# B&R Automation Studio project SuperTrak_Distribution (part 2)

#### HmiWriteParID.st - HmiWriteParID function block
```iecst
(******************************************************************************************
 * Copyright: Bernecker + Rainer
 * Author:  B+R
 * Created:  July 2, 2018/1:30 PM
 ******************************************************************************************
 ******************************************************************************************
 * Version History:
 * ----------------------------------------------------------------------------------------
 * V 1.00.0   July 2, 2018/1:30 PM  First Version
 ******************************************************************************************
 * Description:
 * ----------------------------------------------------------------------------------------
 * July 2, 2018/1:30 PM V1.00.0:
 * This FUNCTION block writes ParIDs TO the SuperTrak.
 * Additionally a parameter save can be executed.
 * The FUB can be connected directly TO a HMI application.
 * The parameter structure AND I/Os can be used inside the visu without extra implementation.
 ******************************************************************************************)

FUNCTION_BLOCK HMIWriteParID

	// Check if function block is enabled
	IF Enable THEN
		//####################################################################################//
		// FUNCTION BLOCK IS ENABLED
		//####################################################################################//

		// Check if error occured to change state
		IF Error THEN
			// Go to state error, to wait for acknowledge
			Internal.Step																	:= HMI_WPAR_STATE_ERROR;
		END_IF;

		//************************************************************************************//
		// Operation
		//************************************************************************************//
		CASE Internal.Step OF
			//--------------------------------------------------------------------------------//
			// Initialize internal parameters
			//--------------------------------------------------------------------------------//
			HMI_WPAR_STATE_INIT:

				// Initialize function block to create a logbook entry
				Internal.ArEventLogWrite.AddData											:= ADR(Internal.AddErrorInfo);
				Internal.ArEventLogWrite.AddDataFormat										:= 1;	// zero-terminated string
				Internal.ArEventLogWrite.AddDataSize										:= SIZEOF(Internal.AddErrorInfo);
				Internal.ArEventLogWrite.ObjectID											:= 'HMIWriteParID';
				Internal.AddErrorInfo														:= '';
				Internal.ArEventLogWrite.OriginRecordID										:= 0;	// don't use origin record
				Internal.ArEventLogWrite.TimeStamp											:= 0;	// use internal time stamp

				Internal.Step																:= HMI_WPAR_STATE_INIT_CHECK_CONFIG;

				//--------------------------------------------------------------------------------//
				// Register function block
				//--------------------------------------------------------------------------------//
			HMI_WPAR_STATE_INIT_CHECK_CONFIG:

				// Check configuration inputs if valid
				IF (ADR(Parameters) > 0) AND
					(ADR(HMILink) > 0) THEN
					// Config OK
					Internal.Status.InitConfigCheckDone										:= TRUE;
					Internal.Step															:= HMI_WPAR_STATE_INIT_REG_FB;
				ELSE
					Internal.Status.InitConfigCheckDone										:= FALSE;
					// Set error
					StatusID																:= HMI_ERR_WRONG_CONFIG;
					Error																	:= TRUE;
				END_IF;

				//--------------------------------------------------------------------------------//
				// Register function block
				//--------------------------------------------------------------------------------//
			HMI_WPAR_STATE_INIT_REG_FB:

				// Check if function block is not registered yet
				IF NOT Internal.Status.FuncitonBlockRegistered THEN
					// Check if StControl instance is present and valid
					IF (HMILink.LibraryStatus.FbID[0] <> 0) AND (HMILink.LibraryStatus.LogBookIdent <> 0) THEN
						// Save logbook ident
						Internal.ArEventLogWrite.Ident										:= HMILink.LibraryStatus.LogBookIdent;
						// Create function block ID
						Internal.Status.FuncitonBlockID										:= HMI_CONFIG_FB_ID_HMIWRITE;
						Internal.Status.FunctionBlockIDIndex								:= 0;
						Internal.Status.FuncitonBlockRegistered								:= TRUE;
						// Create logbook entry
						Internal.AddErrorInfo												:= 'Function block registration successfull';
						Internal.ArEventLogWrite.EventID									:= HMI_SUCC_FB_REGISTRATION;
						// Write logbook entry
						WriteLogbookEntry;
					ELSIF (HMILink.LibraryStatus.LogBookIdent <> 0) THEN
						Internal.AddErrorInfo												:= 'No enabled instance of HMIControl could be found';
						Internal.ArEventLogWrite.EventID									:= HMI_ERR_NO_HMICONTROL_REG;
						// Write logbook entry
						WriteLogbookEntry;
						// Set error
						StatusID															:= HMI_ERR_NO_HMICONTROL_REG;
						Error																:= TRUE;
					ELSE
						// Set error
						StatusID															:= HMI_ERR_NO_HMICONTROL_REG;
						Error																:= TRUE;
					END_IF;
				ELSE
					// Continue
					Internal.Step															:= HMI_WPAR_STATE_INIT_CHECK_PAR;
				END_IF;

				//--------------------------------------------------------------------------------//
				// Check parameters
				//--------------------------------------------------------------------------------//
			HMI_WPAR_STATE_INIT_CHECK_PAR:

				// Save parameters
				Internal.ParametersUsed														:= Parameters;
				Internal.Status.InitParCheckDone											:= TRUE;
				Internal.Step																:= HMI_WPAR_STATE_OPERATION;

				//--------------------------------------------------------------------------------//
				// Operation
				//--------------------------------------------------------------------------------//
			HMI_WPAR_STATE_OPERATION:

				// Set active output
				Active																		:= TRUE;

				// Check configuration inputs if valid
				IF (ADR(Parameters) > 0) AND
					(ADR(HMILink) > 0) THEN
					//:::::::::::::::::::::::::::::::::::::::::::::::::::::::::::::::::::::::::::://
					// Parameter update handling
					// Check if parameters should be updated
					IF Update AND NOT Internal.UpdateOld AND NOT UpdateDone THEN

						// Check if parameters are valid
						IF (Parameters.ParameterNumber <> 0) AND
							(Parameters.SectionID <= HMI_CONFIG_NR_OF_SECTIONS) THEN
							// PARAMTERS ARE VALID
							// copy paramters to internal stucture
							Internal.ParametersUsed												:= Parameters;
							// Set status output that update is done
							UpdateDone															:= TRUE;
						ELSE
							// PARAMTERS ARE INVALID
							IF (Parameters.ParameterNumber = 0) THEN
								Internal.AddErrorInfo											:= 'Parameter ID is invalid';
							ELSIF (Parameters.SectionID > HMI_CONFIG_NR_OF_SECTIONS) THEN
								Internal.AddErrorInfo											:= 'Number of section is invalid';
							END_IF;
							Internal.ArEventLogWrite.EventID									:= HMI_ERR_WRONG_PARAMETER;
							// Write logbook entry
							WriteLogbookEntry;
							// Set error
							StatusID															:= HMI_ERR_WRONG_PARAMETER;
							Error																:= TRUE;
						END_IF;
					ELSIF NOT Update THEN
						UpdateDone																:= FALSE;
					END_IF;

					//:::::::::::::::::::::::::::::::::::::::::::::::::::::::::::::::::::::::::::://
					// Service Channel implementation
					// Check if paramter should be written
					IF WriteUDINT AND NOT(CommandDone) THEN
						// Check if parameters are valid
						IF (Parameters.ParameterNumber <> 0) AND
							(Parameters.SectionID <= HMI_CONFIG_NR_OF_SECTIONS) THEN
							// PARAMTERS ARE VALID
							// copy paramters to internal stucture
							Internal.ParametersUsed												:= Parameters;
							Internal.Status.WriteStatus := SuperTrakServChanWrite(Parameters.SectionID,Parameters.ParameterNumber,Parameters.StartParameterIndex,Parameters.ParameterValueCount,ADR(Parameters.UDINTvalue),SIZEOF(Parameters.UDINTvalue));
							IF Internal.Status.WriteStatus <> 0 THEN
								Internal.AddErrorInfo											:= 'Command was not executed successfully: ';
								Info.ErrorCode													:= Internal.Status.WriteStatus;
								GetErrorCode;
								Internal.ArEventLogWrite.EventID								:= HMI_ERR_CMD_NOT_EXECUTED;
								// Write logbook entry
								WriteLogbookEntry;
								// Set error
								StatusID														:= HMI_ERR_CMD_NOT_EXECUTED;
								Error															:= TRUE;
							ELSE
								CommandDone														:= TRUE;
							END_IF;
						ELSE
							// PARAMTERS ARE INVALID
							IF (Parameters.ParameterNumber = 0) THEN
								Internal.AddErrorInfo											:= 'Parameter ID is invalid';
							ELSIF (Parameters.SectionID > HMI_CONFIG_NR_OF_SECTIONS) THEN
								Internal.AddErrorInfo											:= 'Number of section is invalid';
							END_IF;
							Internal.ArEventLogWrite.EventID									:= HMI_ERR_WRONG_PARAMETER;
							// Write logbook entry
							WriteLogbookEntry;
							// Set error
							StatusID															:= HMI_ERR_WRONG_PARAMETER;
							Error																:= TRUE;
						END_IF;

					ELSIF WriteUINT AND NOT(CommandDone) THEN
							// Check if parameters are valid
							IF (Parameters.ParameterNumber <> 0) AND
								(Parameters.SectionID <= HMI_CONFIG_NR_OF_SECTIONS) THEN
								// PARAMTERS ARE VALID
								// copy paramters to internal stucture
								Internal.ParametersUsed												:= Parameters;
								Internal.Status.WriteStatus := SuperTrakServChanWrite(Parameters.SectionID,Parameters.ParameterNumber,Parameters.StartParameterIndex,Parameters.ParameterValueCount,ADR(Parameters.UINTvalue),SIZEOF(Parameters.UINTvalue));
								IF Internal.Status.WriteStatus <> 0 THEN
									Internal.AddErrorInfo											:= 'Command was not executed successfully: ';
									Info.ErrorCode													:= Internal.Status.WriteStatus;
									GetErrorCode;
									Internal.ArEventLogWrite.EventID								:= HMI_ERR_CMD_NOT_EXECUTED;
									// Write logbook entry
									WriteLogbookEntry;
									// Set error
									StatusID														:= HMI_ERR_CMD_NOT_EXECUTED;
									Error															:= TRUE;
								ELSE
									CommandDone														:= TRUE;
								END_IF;
							ELSE
								// PARAMTERS ARE INVALID
								IF (Parameters.ParameterNumber = 0) THEN
									Internal.AddErrorInfo											:= 'Parameter ID is invalid';
								ELSIF (Parameters.SectionID > HMI_CONFIG_NR_OF_SECTIONS) THEN
									Internal.AddErrorInfo											:= 'Number of section is invalid';
								END_IF;
								Internal.ArEventLogWrite.EventID									:= HMI_ERR_WRONG_PARAMETER;
								// Write logbook entry
								WriteLogbookEntry;
								// Set error
								StatusID															:= HMI_ERR_WRONG_PARAMETER;
								Error																:= TRUE;
							END_IF;

					ELSIF WriteUSINT AND NOT(CommandDone) THEN
						// Check if parameters are valid
						IF (Parameters.ParameterNumber <> 0) AND
							(Parameters.SectionID <= HMI_CONFIG_NR_OF_SECTIONS) THEN
							// PARAMTERS ARE VALID
							// copy paramters to internal stucture
							Internal.ParametersUsed												:= Parameters;
							Internal.Status.WriteStatus := SuperTrakServChanWrite(Parameters.SectionID,Parameters.ParameterNumber,Parameters.StartParameterIndex,Parameters.ParameterValueCount,ADR(Parameters.USINTvalue),SIZEOF(Parameters.USINTvalue));
							IF Internal.Status.WriteStatus <> 0 THEN
								Internal.AddErrorInfo											:= 'Command was not executed successfully: ';
								Info.ErrorCode													:= Internal.Status.WriteStatus;
								GetErrorCode;
								Internal.ArEventLogWrite.EventID								:= HMI_ERR_CMD_NOT_EXECUTED;
								// Write logbook entry
								WriteLogbookEntry;
								// Set error
								StatusID														:= HMI_ERR_CMD_NOT_EXECUTED;
								Error															:= TRUE;
							ELSE
								CommandDone														:= TRUE;
							END_IF;
						ELSE
							// PARAMTERS ARE INVALID
							IF (Parameters.ParameterNumber = 0) THEN
								Internal.AddErrorInfo											:= 'Parameter ID is invalid';
							ELSIF (Parameters.SectionID > HMI_CONFIG_NR_OF_SECTIONS) THEN
								Internal.AddErrorInfo											:= 'Number of section is invalid';
							END_IF;
							Internal.ArEventLogWrite.EventID									:= HMI_ERR_WRONG_PARAMETER;
							// Write logbook entry
							WriteLogbookEntry;
							// Set error
							StatusID															:= HMI_ERR_WRONG_PARAMETER;
							Error																:= TRUE;
						END_IF;

					ELSIF WriteDINT AND NOT(CommandDone) THEN
						// Check if parameters are valid
						IF (Parameters.ParameterNumber <> 0) AND
							(Parameters.SectionID <= HMI_CONFIG_NR_OF_SECTIONS) THEN
							// PARAMTERS ARE VALID
							// copy paramters to internal stucture
							Internal.ParametersUsed												:= Parameters;
							Internal.Status.WriteStatus := SuperTrakServChanWrite(Parameters.SectionID,Parameters.ParameterNumber,Parameters.StartParameterIndex,Parameters.ParameterValueCount,ADR(Parameters.DINTvalue),SIZEOF(Parameters.DINTvalue));
							IF Internal.Status.WriteStatus <> 0 THEN
								Internal.AddErrorInfo											:= 'Command was not executed successfully: ';
								Info.ErrorCode													:= Internal.Status.WriteStatus;
								GetErrorCode;
								Internal.ArEventLogWrite.EventID								:= HMI_ERR_CMD_NOT_EXECUTED;
								// Write logbook entry
								WriteLogbookEntry;
								// Set error
								StatusID														:= HMI_ERR_CMD_NOT_EXECUTED;
								Error															:= TRUE;
							ELSE
								CommandDone														:= TRUE;
							END_IF;
						ELSE
							// PARAMTERS ARE INVALID
							IF (Parameters.ParameterNumber = 0) THEN
								Internal.AddErrorInfo											:= 'Parameter ID is invalid';
							ELSIF (Parameters.SectionID > HMI_CONFIG_NR_OF_SECTIONS) THEN
								Internal.AddErrorInfo											:= 'Number of section is invalid';
							END_IF;
							Internal.ArEventLogWrite.EventID									:= HMI_ERR_WRONG_PARAMETER;
							// Write logbook entry
							WriteLogbookEntry;
							// Set error
							StatusID															:= HMI_ERR_WRONG_PARAMETER;
							Error																:= TRUE;
						END_IF;

					ELSIF WriteINT AND NOT(CommandDone) THEN
						// Check if parameters are valid
						IF (Parameters.ParameterNumber <> 0) AND
							(Parameters.SectionID <= HMI_CONFIG_NR_OF_SECTIONS) THEN
							// PARAMTERS ARE VALID
							// copy paramters to internal stucture
							Internal.ParametersUsed												:= Parameters;
							Internal.Status.WriteStatus := SuperTrakServChanWrite(Parameters.SectionID,Parameters.ParameterNumber,Parameters.StartParameterIndex,Parameters.ParameterValueCount,ADR(Parameters.INTvalue),SIZEOF(Parameters.INTvalue));
							IF Internal.Status.WriteStatus <> 0 THEN
								Internal.AddErrorInfo											:= 'Command was not executed successfully: ';
								Info.ErrorCode													:= Internal.Status.WriteStatus;
								GetErrorCode;
								Internal.ArEventLogWrite.EventID								:= HMI_ERR_CMD_NOT_EXECUTED;
								// Write logbook entry
								WriteLogbookEntry;
								// Set error
								StatusID														:= HMI_ERR_CMD_NOT_EXECUTED;
								Error															:= TRUE;
							ELSE
								CommandDone														:= TRUE;
							END_IF;
						ELSE
							// PARAMTERS ARE INVALID
							IF (Parameters.ParameterNumber = 0) THEN
								Internal.AddErrorInfo											:= 'Parameter ID is invalid';
							ELSIF (Parameters.SectionID > HMI_CONFIG_NR_OF_SECTIONS) THEN
								Internal.AddErrorInfo											:= 'Number of section is invalid';
							END_IF;
							Internal.ArEventLogWrite.EventID									:= HMI_ERR_WRONG_PARAMETER;
							// Write logbook entry
							WriteLogbookEntry;
							// Set error
							StatusID															:= HMI_ERR_WRONG_PARAMETER;
							Error																:= TRUE;
						END_IF;

					ELSIF WriteSINT AND NOT(CommandDone) THEN
						// Check if parameters are valid
						IF (Parameters.ParameterNumber <> 0) AND
							(Parameters.SectionID <= HMI_CONFIG_NR_OF_SECTIONS) THEN
							// PARAMTERS ARE VALID
							// copy paramters to internal stucture
							Internal.ParametersUsed												:= Parameters;
							Internal.Status.WriteStatus := SuperTrakServChanWrite(Parameters.SectionID,Parameters.ParameterNumber,Parameters.StartParameterIndex,Parameters.ParameterValueCount,ADR(Parameters.SINTvalue),SIZEOF(Parameters.SINTvalue));
							IF Internal.Status.WriteStatus <> 0 THEN
								Internal.AddErrorInfo											:= 'Command was not executed successfully: ';
								Info.ErrorCode													:= Internal.Status.WriteStatus;
								GetErrorCode;
								Internal.ArEventLogWrite.EventID								:= HMI_ERR_CMD_NOT_EXECUTED;
								// Write logbook entry
								WriteLogbookEntry;
								// Set error
								StatusID														:= HMI_ERR_CMD_NOT_EXECUTED;
								Error															:= TRUE;
							ELSE
								CommandDone														:= TRUE;
							END_IF;
						ELSE
							// PARAMTERS ARE INVALID
							IF (Parameters.ParameterNumber = 0) THEN
								Internal.AddErrorInfo											:= 'Parameter ID is invalid';
							ELSIF (Parameters.SectionID > HMI_CONFIG_NR_OF_SECTIONS) THEN
								Internal.AddErrorInfo											:= 'Number of section is invalid';
							END_IF;
							Internal.ArEventLogWrite.EventID									:= HMI_ERR_WRONG_PARAMETER;
							// Write logbook entry
							WriteLogbookEntry;
							// Set error
							StatusID															:= HMI_ERR_WRONG_PARAMETER;
							Error																:= TRUE;
						END_IF;

					ELSIF WriteREAL AND NOT(CommandDone) THEN
						// Check if parameters are valid
						IF (Parameters.ParameterNumber <> 0) AND
							(Parameters.SectionID <= HMI_CONFIG_NR_OF_SECTIONS) THEN
							// PARAMTERS ARE VALID
							// copy paramters to internal stucture
							Internal.ParametersUsed												:= Parameters;
							Internal.Status.WriteStatus := SuperTrakServChanWrite(Parameters.SectionID,Parameters.ParameterNumber,Parameters.StartParameterIndex,Parameters.ParameterValueCount,ADR(Parameters.REALvalue),SIZEOF(Parameters.REALvalue));
							IF Internal.Status.WriteStatus <> 0 THEN
								Internal.AddErrorInfo											:= 'Command was not executed successfully: ';
								Info.ErrorCode													:= Internal.Status.WriteStatus;
								GetErrorCode;
								Internal.ArEventLogWrite.EventID								:= HMI_ERR_CMD_NOT_EXECUTED;
								// Write logbook entry
								WriteLogbookEntry;
								// Set error
								StatusID														:= HMI_ERR_CMD_NOT_EXECUTED;
								Error															:= TRUE;
							ELSE
								CommandDone														:= TRUE;
							END_IF;
						ELSE
							// PARAMTERS ARE INVALID
							IF (Parameters.ParameterNumber = 0) THEN
								Internal.AddErrorInfo											:= 'Parameter ID is invalid';
							ELSIF (Parameters.SectionID > HMI_CONFIG_NR_OF_SECTIONS) THEN
								Internal.AddErrorInfo											:= 'Number of section is invalid';
							END_IF;
							Internal.ArEventLogWrite.EventID									:= HMI_ERR_WRONG_PARAMETER;
							// Write logbook entry
							WriteLogbookEntry;
							// Set error
							StatusID															:= HMI_ERR_WRONG_PARAMETER;
							Error																:= TRUE;
						END_IF;

					ELSIF WriteSTRING AND NOT(CommandDone) THEN
						// Check if parameters are valid
						IF (Parameters.ParameterNumber <> 0) AND
							(Parameters.SectionID <= HMI_CONFIG_NR_OF_SECTIONS) AND
							(Parameters.STRINGsize > 0) THEN
							// PARAMTERS ARE VALID
							// copy paramters to internal stucture
							Internal.ParametersUsed												:= Parameters;
							Internal.Status.WriteStatus := SuperTrakServChanWrite(Parameters.SectionID,Parameters.ParameterNumber,Parameters.StartParameterIndex,Parameters.STRINGsize,ADR(Parameters.STRINGvalue),Parameters.STRINGsize);
							IF Internal.Status.WriteStatus <> 0 THEN
								Internal.AddErrorInfo											:= 'Command was not executed successfully: ';
								Info.ErrorCode													:= Internal.Status.WriteStatus;
								GetErrorCode;
								Internal.ArEventLogWrite.EventID								:= HMI_ERR_CMD_NOT_EXECUTED;
								// Write logbook entry
								WriteLogbookEntry;
								// Set error
								StatusID														:= HMI_ERR_CMD_NOT_EXECUTED;
								Error															:= TRUE;
							ELSE
								CommandDone														:= TRUE;
							END_IF;
						ELSE
							// PARAMTERS ARE INVALID
							IF (Parameters.ParameterNumber = 0) THEN
								Internal.AddErrorInfo											:= 'Parameter ID is invalid';
							ELSIF (Parameters.SectionID > HMI_CONFIG_NR_OF_SECTIONS) THEN
								Internal.AddErrorInfo											:= 'Number of section is invalid';
							END_IF;
							Internal.ArEventLogWrite.EventID									:= HMI_ERR_WRONG_PARAMETER;
							// Write logbook entry
							WriteLogbookEntry;
							// Set error
							StatusID															:= HMI_ERR_WRONG_PARAMETER;
							Error																:= TRUE;
						END_IF;

						// Check if paramters should be saved
					ELSIF SaveParameters AND NOT(CommandDone) THEN
						Internal.SaveValue	:= 0;

						IF Parameters.Save.SystemLayout THEN
							Internal.SaveValue := BIT_SET(Internal.SaveValue,1);
						END_IF;
						IF Parameters.Save.Targets THEN
							Internal.SaveValue := BIT_SET(Internal.SaveValue,2);
						END_IF;
						IF Parameters.Save.Regions THEN
							Internal.SaveValue := BIT_SET(Internal.SaveValue,3);
						END_IF;
						IF Parameters.Save.MoveConfig THEN
							Internal.SaveValue := BIT_SET(Internal.SaveValue,4);
						END_IF;
						IF Parameters.Save.GlobalPar THEN
							Internal.SaveValue := BIT_SET(Internal.SaveValue,5);
						END_IF;
						IF Parameters.Save.Offsets THEN
							Internal.SaveValue := BIT_SET(Internal.SaveValue,6);
						END_IF;
						IF Parameters.Save.SectionPar THEN
							Internal.SaveValue := BIT_SET(Internal.SaveValue,9);
						END_IF;
						IF Parameters.Save.ControlGains THEN
							Internal.SaveValue := BIT_SET(Internal.SaveValue,11);
						END_IF;
						IF Parameters.Save.EncoderConfig THEN
							Internal.SaveValue := BIT_SET(Internal.SaveValue,12);
						END_IF;
						IF Parameters.Save.IRTagConfig THEN
							Internal.SaveValue := BIT_SET(Internal.SaveValue,13);
						END_IF;
						IF Parameters.Save.VirtualIO THEN
							Internal.SaveValue := BIT_SET(Internal.SaveValue,14);
						END_IF;
						IF Parameters.Save.PosTrig THEN
							Internal.SaveValue := BIT_SET(Internal.SaveValue,15);
						END_IF;

						Internal.Status.WriteStatus := SuperTrakServChanWrite(0,HMI_SC_SAVE_PARAMTER_CODE,0,1,ADR(Internal.SaveValue),SIZEOF(Internal.SaveValue));
						IF Internal.Status.WriteStatus <> 0 THEN
							Internal.AddErrorInfo											:= 'Command was not executed successfully: ';
							Info.ErrorCode													:= Internal.Status.WriteStatus;
							GetErrorCode;
							Internal.ArEventLogWrite.EventID								:= HMI_ERR_CMD_NOT_EXECUTED;
							// Write logbook entry
							WriteLogbookEntry;
							// Set error
							StatusID														:= HMI_ERR_CMD_NOT_EXECUTED;
							Error															:= TRUE;
						ELSE
							CommandDone														:= TRUE;
						END_IF;
					END_IF;

					IF NOT(WriteUDINT) AND NOT(WriteUINT) AND NOT(WriteUSINT) AND NOT(WriteDINT) AND NOT(WriteINT) AND NOT(WriteSINT) AND NOT(WriteREAL) AND NOT(WriteSTRING) AND NOT(SaveParameters) THEN
						CommandDone	:= FALSE;
					END_IF;

					//:::::::::::::::::::::::::::::::::::::::::::::::::::::::::::::::::::::::::::://
					// Error detection
					// Check if communication is not established
					IF NOT HMILink.SuperTrakStatus.StatusValid THEN
						IF (HMILink.LibraryStatus.FbID[0] = 0) AND (HMILink.LibraryStatus.LogBookIdent <> 0) THEN
							Internal.AddErrorInfo												:= 'No enabled instance of HMIControl could be found';
							Internal.ArEventLogWrite.EventID									:= HMI_ERR_NO_HMICONTROL_REG;
							// Write logbook entry
							WriteLogbookEntry;
							// Set error
							StatusID															:= HMI_ERR_NO_HMICONTROL_REG;
							Error																:= TRUE;
						ELSE
							// Set error
							Internal.AddErrorInfo												:= 'No communication to SuperTrak';
							Internal.ArEventLogWrite.EventID									:= HMI_ERR_COMMUNICAITON_TIME_OUT;
							// Write logbook entry
							WriteLogbookEntry;
							StatusID															:= HMI_ERR_COMMUNICAITON_TIME_OUT;
							Error																:= TRUE;
						END_IF;
					END_IF;
				ELSE
					Internal.Status.InitConfigCheckDone											:= FALSE;
					// Set error
					StatusID																	:= HMI_ERR_WRONG_CONFIG;
					Error																		:= TRUE;
				END_IF;

			//--------------------------------------------------------------------------------//
			// Error handling
			//--------------------------------------------------------------------------------//
			HMI_WPAR_STATE_ERROR:

				// Reset active output
				Active																		:= FALSE;

				UpdateDone																	:= FALSE;
				CommandDone																	:= FALSE;

				IF NOT Error THEN
					// Check in which state to jump
					IF NOT Internal.Status.FuncitonBlockRegistered THEN
						Internal.Step														:= HMI_WPAR_STATE_INIT;
					ELSIF NOT Internal.Status.InitConfigCheckDone THEN
						Internal.Step														:= HMI_WPAR_STATE_INIT;
					ELSIF NOT Internal.Status.InitParCheckDone THEN
						Internal.Step														:= HMI_WPAR_STATE_INIT_CHECK_PAR;
					ELSE
						Internal.Step														:= HMI_WPAR_STATE_OPERATION;
					END_IF;
				END_IF;

		END_CASE;

		//************************************************************************************//
		// Error and Warning acknowledgement
		//************************************************************************************//

		// Check if error or warning is acknowledged by user
		IF ErrorReset AND Error AND NOT Internal.ErrorResetOld THEN
			// Reset error
			StatusID																		:= HMI_NO_ERROR;
			Error																			:= FALSE;
			Internal.Status.WriteStatus														:= 0;
			Info.ErrorCode																	:= 0;
		ELSIF ErrorReset AND StatusID <> HMI_NO_ERROR AND NOT Internal.ErrorResetOld THEN
			// Reset warning
			StatusID																		:= HMI_NO_ERROR;
			Internal.Status.WriteStatus														:= 0;
			Info.ErrorCode																	:= 0;
		END_IF;

		// Copy command for edge detection
		Internal.ErrorResetOld																:= ErrorReset;
		Internal.UpdateOld																	:= Update;

	ELSE
		//####################################################################################//
		// FUNCTION BLOCK IS DISABLED
		//####################################################################################//
		// Reset all outputs
		Active																				:= FALSE;
		Error																				:= FALSE;
		StatusID																			:= 0;
		UpdateDone																			:= FALSE;

		CommandDone																			:= FALSE;

		Internal.Status.FuncitonBlockRegistered												:= FALSE;
		Internal.Status.InitParCheckDone													:= FALSE;
		Internal.Status.InitConfigCheckDone													:= FALSE;
		Internal.Step																		:= HMI_WPAR_STATE_INIT;

		Internal.Status.WriteStatus															:= 0;
		Info.ErrorCode																		:= 0;
	END_IF;

END_FUNCTION_BLOCK
```

#### GlobalActions.st - The actions defined here are used in the function block implementations
```iecst
(******************************************************************************************
 * Copyright: Bernecker + Rainer
 * Author:  B+R
 * Created:  July 2, 2018/10:07 AM
 ******************************************************************************************
 ******************************************************************************************
 * Version History:
 * ----------------------------------------------------------------------------------------
 * V 1.00.0   July 2, 2018/10:07 AM  First Version
 ******************************************************************************************
 * Description:
 * ----------------------------------------------------------------------------------------
 * July 2, 2018/10:07 AM V1.00.0:
 * The actions defined here are used in the FUNCTION block implementations.
 * All FUNCTION blocks, where these actions should be used, must have the
 * variables used here as part OF the internal structure
 ******************************************************************************************)

ACTION WriteLogbookEntry:

	// Set command to write logbook entry
	Internal.ArEventLogWrite.Execute						:= TRUE;
	// Function block call
	Internal.ArEventLogWrite();
	// Check if writing of logbook entry is finished, to reset command
	IF Internal.ArEventLogWrite.Done THEN
		// Reset additional error info
		brsmemset(ADR(Internal.AddErrorInfo), 0, SIZEOF(Internal.AddErrorInfo));
		// Reset command to create logbook entry
		Internal.ArEventLogWrite.Execute					:= FALSE;
		// Function block call
		Internal.ArEventLogWrite();
	ELSIF Internal.ArEventLogWrite.Error THEN
		// Set command to write logbook entry
		Internal.ArEventLogWrite.Execute					:= FALSE;
		// Function block call
		Internal.ArEventLogWrite();
		StatusID											:= Internal.ArEventLogWrite.StatusID;
		Error												:= TRUE;
	END_IF;

END_ACTION

ACTION GetErrorCode:

	CASE Info.ErrorCode OF
		1:
			brsstrcat(ADR(Internal.AddErrorInfo),ADR('An invalid section number was specified.'));

		2:
			brsstrcat(ADR(Internal.AddErrorInfo),ADR('The specified parameter number was not recognized.'));

		3:
			brsstrcat(ADR(Internal.AddErrorInfo),ADR('The specified task code was not recognized.'));

		4:
			brsstrcat(ADR(Internal.AddErrorInfo),ADR('The requested operation is currently unavailable.'));

		6:
			brsstrcat(ADR(Internal.AddErrorInfo),ADR('The specified starting index is invalid.'));

		7:
			brsstrcat(ADR(Internal.AddErrorInfo),ADR('The value to be written was outside of the valid range.'));

		8:
			brsstrcat(ADR(Internal.AddErrorInfo),ADR('The requested number of elements is invalid.'));

		10:
			brsstrcat(ADR(Internal.AddErrorInfo),ADR('The command did not complete in a timely manner.'));

		11:
			brsstrcat(ADR(Internal.AddErrorInfo),ADR('The request was denied due to a lack of permissions.'));

		14:
			brsstrcat(ADR(Internal.AddErrorInfo),ADR('The packet is malformed, or its length is incorrect.'));

		15:
			brsstrcat(ADR(Internal.AddErrorInfo),ADR('An internal error occurred while processing the request.'));

	END_CASE;

END_ACTION
```

### Package Logical/Source - Source code

### Package Logical/Source/SuperTrak - Control the SuperTrak

### Program Logical/Source/SuperTrak/ST_Logic (IEC)

#### Main.st - Init, cyclic, exit code
```iecst
(*********************************************************************************
 * Copyright: Bernecker + Rainer
 * Author:  B+R
 * Created:  July 27, 2016/10:44 AM
 *********************************************************************************
 *********************************************************************************
 * Version History:
 * -------------------------------------------------------------------------------
 * V 1.00.0   July 27, 2016/10:44 AM  First Version
 *********************************************************************************
 * Description:
 * -------------------------------------------------------------------------------
 * July 27, 2016/10:44 AM V1.00.0:
 * This task is an example OF simple SuperTrak control
 *********************************************************************************)

PROGRAM _INIT

 	(*************************************************************************************************)
 	(*************************************************************************************************)
 	(* FUNCTION BLOCK CONFIGURATION *)

 	// Configure the internal communication structure to/from SuperTrak
	SuperTrakControlParameters.NrOfCommands 	:= CONFIG_ST_MAX_COMMANDS;
	SuperTrakControlParameters.NrOfPallets  	:= CONFIG_ST_MAX_PALLETS;
	SuperTrakControlParameters.NrOfSections 	:= CONFIG_ST_MAX_SECTIONS;
	SuperTrakControlParameters.NrOfTargets  	:= CONFIG_ST_MAX_TARGETS;

	(*************************************************************************************************)
	(*************************************************************************************************)
	(* FUNCTION BLOCK INITIALIZATION *)

	// Initialize the function block, handling the communication to/from SuperTrak
	StControl_0.StLink      	 				:= ADR(gStLink);
	StControl_0.Enable       					:= TRUE;
	StControl_0.Parameters      				:= ADR(SuperTrakControlParameters);
	StControl_0.StCtrlData      				:= ADR(gStCyclicControlData);
	StControl_0.StCtrlDataSize     				:= SIZEOF(gStCyclicControlData);
	StControl_0.StStatData      				:= ADR(gStCyclicStatusData);
	StControl_0.StStatDataSize     				:= SIZEOF(gStCyclicStatusData);
	StControl_0.StServChRequestData   			:= ADR(gStServiceChannelReqData);
	StControl_0.StServChRequestDataSize  		:= SIZEOF(gStServiceChannelReqData);
	StControl_0.StServChResponseData  			:= ADR(gStServiceChannelResData);
	StControl_0.StServChResponseDataSize 		:= SIZEOF(gStServiceChannelResData);

	// Initialize the fucntion blocks, controlling a single section
	FOR Index := 0 TO (SIZEOF(StSection_) / SIZEOF(StSection_[0])) - 1 DO
		StSection_[Index].StLink    			:= ADR(gStLink);
		StSection_[Index].Parameters   			:= ADR(SuperTrakSectionParameters);
		StSection_[Index].Section    			:= Index + 1;
	END_FOR;

	// Initialize the fucntion blocks, controlling a single section
	FOR Index := 0 TO (SIZEOF(StTargetExt_) / SIZEOF(StTargetExt_[0])) - 1 DO
		StTargetExt_[Index].StLink    			:= ADR(gStLink);
		StTargetExt_[Index].Parameters  		:= ADR(TargetControlParameters[Index]);
		StTargetExt_[Index].Target    			:= Index + 1;
	END_FOR;

// Initialize the fucntion blocks, controlling a single section
	FOR Index := 0 TO (SIZEOF(StPallet_) / SIZEOF(StPallet_[0])) - 1 DO
		StPallet_[Index].StLink 				:= ADR(gStLink);
		StPallet_[Index].Parameters 			:= ADR(PalletControlParameters[Index]);
		StPallet_[Index].PalletID 				:= Index + 1;

		PalletControlParameters[Index].PalletConfig.Shelf.ShelfWidth					:= 152;
		PalletControlParameters[Index].PalletConfig.Shelf.OffsetFromCenter				:= 0;
		PalletControlParameters[Index].PalletConfig.Controller.ControlGainSetIdx		:= 0;
		PalletControlParameters[Index].PalletConfig.Controller.FilterWeightMoving		:= 0.5;
		PalletControlParameters[Index].PalletConfig.Controller.FilterWeightStationary	:= 0.5;
	END_FOR;

	// Initialize the function block for AntiSloshing
	StAdvCmd_0.StLink 							:= ADR(gStLink);
	StAdvCmd_0.Parameters 						:= ADR(StAdvCmdParameters);

	// Set Parameters for AntiSloshing
	StAdvCmdParameters.CommandID   	 			:= 82;				// Specify the Control-Parent; 80 -> Target; 82 -> PalletID
	StAdvCmdParameters.Context		 			:= 1;				// Used PalletID -> 1; ID will be checked at the start of the Anti-Sloshing mode
	StAdvCmdParameters.Parameters[0] 			:= 1;				// Used Container-Shape; 0 -> None; 1 -> Rectangle; 2 -> Cylinder
	StAdvCmdParameters.Parameters[1] 			:= 2;				// Used Oscillation-Mode
	StAdvCmdParameters.Parameters[2] 			:= 189;				// Length of the Container [mm], "Liquid-Length"
	StAdvCmdParameters.Parameters[3]			:= 0;
	StAdvCmdParameters.Parameters[4] 			:= 58;				// Fill-Height of the liquid
	StAdvCmdParameters.Parameters[5] 			:= 0;

	ContainerShape								:= 1;				// Used Container-Shape; 0 -> None; 1 -> Rectangle; 2 -> Cylinder
	ContainerLength								:= 189;				// Length of the Container [mm], "Liquid-Length"
	ContainerHeight								:= 58;				// Fill-Height of the liquid

	// Set start parameters to read temperatures
	SectionID									:= 1;

	// Set start section to be displayed at the Temperatures, Alarm and Shuttle page
	VisuSection									:= 1;
	VisuAlarmSection							:= 1;
	VisuShuttle									:= 1;

	// Target where shuttles get IDs
	StartTarget									:= 1;
	WaitTarget									:= 2;

	// Start of the Expert mode
	StateCnc									:= EXPERT_MODE_START;
	CncStartTarget								:= 1;

	// Set the WritePnu parameter
	StWritePnu_Region.StLink					:= ADR(gStLink);
	StWritePnu_Region.Parameters				:= ADR(StWritePnuPar_Region);

	// Set the ReadPnu parameter
	StReadPnu_Region.StLink						:= ADR(gStLink);
	StReadPnu_Region.Parameters					:= ADR(StReadPnuPar_Region);

	RegionStatus								:= 7;			// 7 --> Bit 0,1,2 --> Enable Region, Limit v, Limit a
	TimerRegionEnable.PT						:= T#1s;

	// Get the used cycle time
	RTInfo_0.enable								:= TRUE;
	RTInfo_0();
	CycleTime									:= UDINT_TO_REAL(RTInfo_0.cycle_time)/1000;

	// Init mappAlarmX parameters
	AlarmXInit;

	//ParID Hmi Init
	InitParID;

	// Init shuttle config page
	Config_ShelfWidth				:= 152;
	Config_OffsetFromCenter			:= 0;
	Config_ControlGainSetIndex		:= 0;
	Config_FilterWeightMoving		:= 0.5;
	Config_FilterWeightStationary	:= 0.5;

END_PROGRAM

PROGRAM _CYCLIC

 	(*************************************************************************************************)
 	(*************************************************************************************************)
 	(* FUNCTION BLOCK ENABLE *)

 	// Wait for StControl to be active, before enalbing all other function blocks
	IF StControl_0.Active THEN
		// Loop thru all StSection function blocks
		FOR Index := 0 TO (SIZEOF(StSection_) / SIZEOF(StSection_[0])) - 1 DO
			// Enable StSection
			StSection_[Index].Enable     		:= TRUE;
			IF StSection_[Index].Error = FALSE AND StSection_[Index].Info.SuperTrak.SectionFaultActive = FALSE AND StSection_[Index].ErrorReset THEN
				StSection_[Index].ErrorReset	:= FALSE;
			END_IF;
		END_FOR;

		// Loop thru all StTargetExt function blocks
		FOR Index := 0 TO (SIZEOF(StTargetExt_) / SIZEOF(StTargetExt_[0])) - 1 DO
			// Enable StTargetExt
			StTargetExt_[Index].Enable     		:= TRUE;
			IF StTargetExt_[Index].Error = FALSE AND StTargetExt_[Index].ErrorReset THEN
				StTargetExt_[Index].ErrorReset	:= FALSE;
			END_IF;
		END_FOR;

		// Loop thru all StPallet function blocks
		FOR Index := 0 TO (SIZEOF(StPallet_) / SIZEOF(StPallet_[0])) - 1 DO
			// Enable StPallet
			StPallet_[Index].Enable 			:= TRUE;
			IF StPallet_[Index].Error = FALSE AND StPallet_[Index].ErrorReset THEN
				StPallet_[Index].ErrorReset		:= FALSE;
			END_IF;
		END_FOR;

		// Enable AntiSloshing function block
		StAdvCmd_0.Enable 						:= TRUE;

		// Reset ErrorReset
		IF StReadPnu_Region.Error = FALSE AND StReadPnu_Region.ErrorReset THEN
			StReadPnu_Region.ErrorReset			:= FALSE;
		END_IF;

		// Reset ErrorReset
		IF StWritePnu_Region.Error = FALSE AND StWritePnu_Region.ErrorReset THEN
			StWritePnu_Region.ErrorReset		:= FALSE;
		END_IF;

		// Enable the start-up region
		IF NOT(IDSet) AND RegionEnabled = FALSE THEN
			EnableRegion;
		END_IF;
	END_IF;

	// Wait for HmiControl to be active, before enalbing all other function blocks
	IF HmiControl_0.Active THEN
		HmiWriteParID_0.Enable					:= TRUE;
		HmiReadParID_0.Enable					:= TRUE;

		IF HmiWriteParID_0.SaveParameters AND HmiWriteParID_0.CommandDone THEN
			SaveSuccessful						:= TRUE;
			SaveFailed							:= FALSE;
		ELSIF HmiWriteParID_0.SaveParameters AND HmiWriteParID_0.Error THEN
			SaveSuccessful						:= FALSE;
			SaveFailed							:= TRUE;
		END_IF;

		IF NOT(HmiWriteParID_0.SaveParameters) AND EDGEPOS(HmiWriteParID_0.CommandDone) THEN
			SaveSuccessful						:= FALSE;
			SaveFailed							:= FALSE;
		END_IF;

		IF HmiWriteParID_0.Error THEN
			HmiWriteParID_0.WriteUDINT			:= FALSE;
			HmiWriteParID_0.WriteUINT			:= FALSE;
			HmiWriteParID_0.WriteUSINT			:= FALSE;
			HmiWriteParID_0.WriteDINT			:= FALSE;
			HmiWriteParID_0.WriteINT			:= FALSE;
			HmiWriteParID_0.WriteSINT			:= FALSE;
			HmiWriteParID_0.WriteREAL			:= FALSE;
			HmiWriteParID_0.WriteSTRING			:= FALSE;
			HmiWriteParID_0.SaveParameters		:= FALSE;
		END_IF;

		IF HmiReadParID_0.Error THEN
			HmiReadParID_0.ReadUDINT			:= FALSE;
			HmiReadParID_0.ReadUINT				:= FALSE;
			HmiReadParID_0.ReadUSINT			:= FALSE;
			HmiReadParID_0.ReadDINT				:= FALSE;
			HmiReadParID_0.ReadINT				:= FALSE;
			HmiReadParID_0.ReadSINT				:= FALSE;
			HmiReadParID_0.ReadREAL				:= FALSE;
			HmiReadParID_0.ReadSTRING			:= FALSE;
		END_IF;

		IF HmiReadParID_0.Error = FALSE AND HmiReadParID_0.ErrorReset THEN
			HmiReadParID_0.ErrorReset			:= FALSE;
		END_IF;

		IF HmiWriteParID_0.Error = FALSE AND HmiWriteParID_0.ErrorReset THEN
			HmiWriteParID_0.ErrorReset			:= FALSE;
		END_IF;
	END_IF;

	// Read temperatures
	ReadTemp;

	(*************************************************************************************************)
	(*************************************************************************************************)
	(* ENABLE / DISABLE SUPERTRAK SECTIONS *)

	// Wait for command, to enable all sections
	IF SuperTrakControl.Command.EnableAllSections THEN
		// Loop thru all StSection function blocks
		FOR Index := 0 TO (SIZEOF(StSection_) / SIZEOF(StSection_[0])) - 1 DO
			// Check if section is ready to be enalbed
			IF StSection_[Index].MotorPowerOn AND NOT StSection_[Index].Error THEN
				// Enable section
				StSection_[Index].EnableSection := TRUE;
			END_IF;
		END_FOR;

		// If command is reset, disable all sections
	ELSE
		// Loop thru all StSection function blocks
		FOR Index := 0 TO (SIZEOF(StSection_) / SIZEOF(StSection_[0])) - 1 DO
			// Disable section
			StSection_[Index].EnableSection    	:= FALSE;
		END_FOR;
	END_IF;

	// Sections enabled and SuperTrak ready to perform a movement
	IF SuperTrakControl.Status.AllSectionsEnabled THEN
		// Set global status to true if all sections are enabled
		gAllSectionsEnabled 					:= TRUE;

		// Get the number of shuttles on the SuperTrak
		NumberOfShuttles						:= UINT_TO_USINT(StControl_0.Info.SuperTrak.NrOfPallets);

		// Check if the shuttles are in standstill
		SuperTrakGetPalletInfo(ADR(ShuttleInfo),NumberOfShuttles,FALSE);
		CheckStandstill;

		// Assign Pallet ID to the existing Shuttles
		IF NOT(IDSet) AND RegionEnabled THEN
			SetPalletIDs;
		END_IF;

		// Disable the start-up region
		IF IDSet AND NOT(RegionDisabled) AND ShuttlesStandstill THEN
			DisableRegion;
		END_IF;

		IF IDSet AND RegionDisabled THEN
			(* Call Actions *)
			IF NOT(SuperTrakControl.Status.TrackingEnabled) AND NOT(SuperTrakControl.Status.PalletControl) THEN
				// Action for AntiSloshing
				AntiSloshing;
			ELSE
				cmd_StartAntiSloshing	:= FALSE;
				cmd_StopAntiSloshing	:= FALSE;
			END_IF;

			IF NOT(SuperTrakControl.Status.TrackingEnabled) AND NOT(SuperTrakControl.Status.AntiSloshingEnabled) THEN
				// Action for Shuttle-Control
				PalletControl;
			ELSE
				cmd_StartPalletControl	:= FALSE;
				cmd_StopPalletControl	:= FALSE;
			END_IF;

			IF NOT(SuperTrakControl.Status.PalletControl) AND NOT(SuperTrakControl.Status.AntiSloshingEnabled) THEN
				// Action for Tracking a shuttle
				ExpertMode;
			ELSE
				cmd_StartTracking		:= FALSE;
				cmd_StopTracking		:= FALSE;
			END_IF;

			// Move all shuttles to target 1 when no mode is selected
			IF NOT(SuperTrakControl.Status.PalletControl) AND NOT(SuperTrakControl.Status.TrackingEnabled) AND NOT(SuperTrakControl.Status.AntiSloshingEnabled) THEN

				FOR Index := 1 TO (SIZEOF(TargetControlParameters) / SIZEOF(TargetControlParameters[0])) - 1 DO
					TargetControlParameters[Index].AdvancedReleaseConfig.DestinationTarget := 1;
					TargetControlParameters[Index].AdvancedReleaseConfig.Direction	       := stCOM_DIR_RIGHT;
					IF StTargetExt_[Index].PalletPresent THEN
						StTargetExt_[Index].ReleaseToTarget	:= TRUE;
					ELSE
						StTargetExt_[Index].ReleaseToTarget := FALSE;
					END_IF;
				END_FOR;

			END_IF;
		END_IF;
	ELSIF IDSet THEN
		// Reset the global status if the sections are not enabled
		gAllSectionsEnabled 	:= FALSE;

		cmd_StartAntiSloshing	:= FALSE;
		cmd_StopAntiSloshing	:= TRUE;
		cmd_StartPalletControl	:= FALSE;
		cmd_StopPalletControl	:= TRUE;
		cmd_StartTracking		:= FALSE;
		cmd_StopTracking		:= TRUE;
	END_IF

	(*************************************************************************************************)
	(*************************************************************************************************)
	(* CALL THE ERROR HANDLING *)
	ReadErrorMessages;

	// Reset all active errors and warnings
	IF AcknowledgeAll THEN
		StControl_0.ErrorReset					:= StControl_0.Error OR StControl_0.StatusID <> 0;
		StReadPnu_Region.ErrorReset				:= StReadPnu_Region.Error OR StReadPnu_Region.StatusID <> 0;
		StWritePnu_Region.ErrorReset			:= StWritePnu_Region.Error OR StWritePnu_Region.StatusID <> 0;
		FOR Index := 0 TO (SIZEOF(StTargetExt_) / SIZEOF(StTargetExt_[0])) - 1 DO
			StTargetExt_[Index].ErrorReset   	:= StTargetExt_[Index].Error OR StTargetExt_[Index].StatusID <> 0;
		END_FOR;
		FOR Index := 0 TO (SIZEOF(StSection_) / SIZEOF(StSection_[0])) - 1 DO
			StSection_[Index].ErrorReset  		:= StSection_[Index].Error OR StSection_[Index].StatusID <> 0;
		END_FOR;
		FOR Index := 0 TO (SIZEOF(StPallet_) / SIZEOF(StPallet_[0])) - 1 DO
			StPallet_[Index].ErrorReset			:= StPallet_[Index].Error OR StPallet_[Index].StatusID <> 0;
		END_FOR;
		HmiReadParID_0.ErrorReset				:= HmiReadParID_0.Error OR HmiReadParID_0.StatusID <> 0;
		HmiWriteParID_0.ErrorReset				:= HmiWriteParID_0.Error OR HmiWriteParID_0.StatusID <> 0;
		AcknowledgeAll							:= FALSE;
	END_IF;

	(*************************************************************************************************)
	(*************************************************************************************************)
	(* Reset Read and Write commands *)
	// Reset all write commands
	IF HmiWriteParID_0.CommandDone THEN
		HmiWriteParID_0.WriteUDINT				:= FALSE;
		HmiWriteParID_0.WriteUINT				:= FALSE;
		HmiWriteParID_0.WriteUSINT				:= FALSE;
		HmiWriteParID_0.WriteDINT				:= FALSE;
		HmiWriteParID_0.WriteINT				:= FALSE;
		HmiWriteParID_0.WriteSINT				:= FALSE;
		HmiWriteParID_0.WriteREAL				:= FALSE;
		HmiWriteParID_0.WriteSTRING				:= FALSE;
	END_IF;

	// Reset all read commands
	IF HmiReadParID_0.CommandDone THEN
		HmiReadParID_0.ReadUDINT				:= FALSE;
		HmiReadParID_0.ReadUINT					:= FALSE;
		HmiReadParID_0.ReadUSINT				:= FALSE;
		HmiReadParID_0.ReadDINT					:= FALSE;
		HmiReadParID_0.ReadINT					:= FALSE;
		HmiReadParID_0.ReadSINT					:= FALSE;
		HmiReadParID_0.ReadREAL					:= FALSE;
		HmiReadParID_0.ReadSTRING				:= FALSE;
	END_IF;

	(*************************************************************************************************)
	(*************************************************************************************************)
	(* CALL THE mapp ALARMX ERROR HANDLING *)

	AlarmX;

	(*************************************************************************************************)
	(*************************************************************************************************)
	(* CALL THE shuttle configuration task *)

	ShuttleConfig;

	(*************************************************************************************************)
	(*************************************************************************************************)
	(* FUNCTION BLOCK CALLS *)

	// Call StControl
	StControl_0();

	// Loop thru all StSection function blocks
	FOR Index := 0 TO (SIZEOF(StSection_) / SIZEOF(StSection_[0])) - 1 DO
		// Call StSection
		StSection_[Index]();
	END_FOR;

	// Loop thru all StTargetExt function blocks
	FOR Index := 0 TO (SIZEOF(StTargetExt_) / SIZEOF(StTargetExt_[0])) - 1 DO
		// Call StTargetExt
		StTargetExt_[Index]();
	END_FOR;

	// Loop thru all StPallet function blocks
	FOR Index := 0 TO (SIZEOF(StPallet_) / SIZEOF(StPallet_[0])) - 1 DO
		// Call StPallet
		StPallet_[Index]();
	END_FOR;

	// Call StAdvCmd
	StAdvCmd_0();

	// Call StWritePnu
	StWritePnu_Region();

	// Call StReadPnu
	StReadPnu_Region();

	// Call the Timer
	TimerRegionEnable();

	// Call HmiControl
	HmiControl_0();

	// Call HmiWriteParID
	HmiWriteParID_0();

	// Call HmiReadParID
	HmiReadParID_0();

	(*************************************************************************************************)
	(*************************************************************************************************)
	(* MAPPING OF STATUS VARIABLES *)

	// Set information on wether all sections are enabled or not, to command structure
	SuperTrakControl.Status.AllSectionsEnabled   := StControl_0.SectionsEnabled;

END_PROGRAM

PROGRAM _EXIT

	// Disable the FUB
	StControl_0.Enable	:= FALSE;
	// Call the StControl
	StControl_0();

	// Loop thru all StSection function blocks
	FOR Index := 0 TO (SIZEOF(StSection_) / SIZEOF(StSection_[0])) - 1 DO
		// Disable the FUB
		StSection_[Index].Enable	:= FALSE;
		// Call StSection
		StSection_[Index]();
	END_FOR;

	// Loop thru all StTargetExt function blocks
	FOR Index := 0 TO (SIZEOF(StTargetExt_) / SIZEOF(StTargetExt_[0])) - 1 DO
		// Disable the FUB
		StTargetExt_[Index].Enable	:= FALSE;
		// Call StTargetExt
		StTargetExt_[Index]();
	END_FOR;

	// Loop thru all StPallet function blocks
	FOR Index := 0 TO (SIZEOF(StPallet_) / SIZEOF(StPallet_[0])) - 1 DO
		// Disable the FUB
		StPallet_[Index].Enable		:= FALSE;
		// Call StPallet
		StPallet_[Index]();
	END_FOR;

	// Disable the FUB
	StAdvCmd_0.Enable				:= FALSE;
	// Call StAdvCmd
	StAdvCmd_0();

	// Disable the FUB
	StWritePnu_Region.Enable		:= FALSE;
	// Call StWritePnu
	StWritePnu_Region();

	// Disable the FUB
	StReadPnu_Region.Enable			:= FALSE;
	// Call StReadPnu
	StReadPnu_Region();

	// Disable the FUB
	HmiControl_0.Enable				:= FALSE;
	// Call StHmiControl
	HmiControl_0();

	// Disable the FUB
	HmiWriteParID_0.Enable			:= FALSE;
	// Call StHmiWriteParID
	HmiWriteParID_0();

	// Disable the FUB
	HmiReadParID_0.Enable			:= FALSE;
	// Call StHmiReadParID
	HmiReadParID_0();

END_PROGRAM
```

#### Types.typ - Local data types
```iecst
(************************************************************************************************************************************)
(************************************************************************************************************************************)
(*Structures for SuperTrak control*)

TYPE
	SuperTrakCtrlType : 	STRUCT  (*Control structure for SuperTrak*)
		Command : SuperTrakCtrlCmdType; (*SuperTrak commands*)
		Parameter : SuperTrakCtrlParType; (*SuperTrak parameters*)
		Status : SuperTrakCtrlStatType; (*SuperTrak status*)
	END_STRUCT;
	SuperTrakCtrlCmdType : 	STRUCT  (*Command strucutre for SuperTrak*)
		EnableAllSections : BOOL; (*Command to enable all sections on the system*)
	END_STRUCT;
	SuperTrakCtrlParType : 	STRUCT  (*Parameter structure for SuperTrak*)
		Reserved : BOOL; (*Reserved for future development*)
	END_STRUCT;
	SuperTrakCtrlStatType : 	STRUCT  (*Status strucutre for SuperTrak*)
		AllSectionsEnabled : BOOL; (*Indicating if all sections on the system are enabled*)
		CommandBusy : BOOL; (*SuperTrak busy*)
		AntiSloshingEnabled : BOOL; (*AntiSloshing function active*)
		TrackingEnabled : BOOL; (*Tracking fuction active*)
		PalletControl : BOOL; (*Shuttle control active*)
	END_STRUCT;
END_TYPE

(*Error handling*)

TYPE
	InfoType : 	STRUCT  (*Error information structure*)
		StControl : StControlErrorInfoType; (*Error information structure StControl*)
		StSection : ARRAY[0..CONFIG_ST_MAX_SECTIONS_MINUS_ONE]OF StSectionErrorInfoType; (*Error information structure StSection*)
		StTargetExt : StTargetExtErrorInfoType; (*Error information structure StTargetExt*)
		StPallet : StPalletErrorInfoType; (*Error information structure StPallet*)
		StReadPnu_Region : StReadPnuErrorInfoType; (*Error information structure StReadPnu*)
		StWritePnu_Region : StWritePnuErrorInfoType; (*Error information structure StWritePnu*)
		HmiWriteParID : HmiWriteParIDErrorInfoType; (*Error information structure HmiWriteParID*)
		HmiReadParID : HmiReadParIDErrorInfoType; (*Error information structure HmiReadParID*)
	END_STRUCT;
	StControlErrorInfoType : 	STRUCT  (*Error information structure StControl*)
		StatusID : DINT; (*Status ID of the FUB*)
		Error : ARRAY[0..23]OF DINT; (*Error number*)
		Warning : ARRAY[0..23]OF DINT; (*Warning number*)
		ErrorText : ARRAY[0..23]OF STRING[80]; (*Error text*)
		WarningText : ARRAY[0..23]OF STRING[80]; (*Warning text*)
	END_STRUCT;
	StSectionErrorInfoType : 	STRUCT  (*Error information structure StSection*)
		StatusID : DINT; (*Status ID of the FUB*)
		Error : ARRAY[0..23]OF DINT; (*Error number*)
		Warning : ARRAY[0..23]OF DINT; (*Warning number*)
		ErrorText : ARRAY[0..23]OF STRING[80]; (*Error text*)
		WarningText : ARRAY[0..23]OF STRING[80]; (*Warning text*)
	END_STRUCT;
	StTargetExtErrorInfoType : 	STRUCT  (*Error information structure StTargetExt*)
		StatusID : ARRAY[0..CONFIG_USED_TARGETS_MINUS_ONE]OF DINT; (*StatusID of the FUB*)
		ErrorText : ARRAY[0..CONFIG_USED_TARGETS_MINUS_ONE]OF STRING[80]; (*Error text*)
		WarningText : ARRAY[0..CONFIG_USED_TARGETS_MINUS_ONE]OF STRING[80]; (*Warning text*)
		TargetID : ARRAY[0..CONFIG_USED_TARGETS_MINUS_ONE]OF USINT; (*Target ID*)
	END_STRUCT;
	StPalletErrorInfoType : 	STRUCT  (*Error information structure StTargetExt*)
		StatusID : ARRAY[0..CONFIG_USED_SHUTTLES_MINUS_ONE]OF DINT; (*StatusID of the FUB*)
		ErrorText : ARRAY[0..CONFIG_USED_SHUTTLES_MINUS_ONE]OF STRING[80]; (*Error text*)
		WarningText : ARRAY[0..CONFIG_USED_SHUTTLES_MINUS_ONE]OF STRING[80]; (*Warning text*)
		ShuttleID : ARRAY[0..CONFIG_USED_SHUTTLES_MINUS_ONE]OF USINT; (*Shuttle ID*)
	END_STRUCT;
	StReadPnuErrorInfoType : 	STRUCT  (*Error information structure StReadPnu*)
		StatusID : DINT; (*StatusID of the FUB*)
		ErrorText : STRING[80]; (*Error text*)
	END_STRUCT;
	StWritePnuErrorInfoType : 	STRUCT  (*Error information structure StWritePnu*)
		StatusID : DINT; (*StatusID of the FUB*)
		ErrorText : STRING[80]; (*Error text*)
	END_STRUCT;
	HmiWriteParIDErrorInfoType : 	STRUCT  (*Error information structure HmiWriteParID*)
		StatusID : DINT; (*StatusID of the FUB*)
		ErrorText : STRING[80]; (*Error text*)
	END_STRUCT;
	HmiReadParIDErrorInfoType : 	STRUCT  (*Error information structure HmiReadParID*)
		StatusID : DINT; (*StatusID of the FUB*)
		ErrorText : STRING[80]; (*Error text*)
	END_STRUCT;
END_TYPE

(*Read temperatures*)

TYPE
	TemperaturesType : 	STRUCT  (*Temperatures structure type*)
		Section : ARRAY[1..CONFIG_ST_MAX_SECTIONS]OF SectionType; (*Section information type*)
	END_STRUCT;
	RealSectionType : 	STRUCT  (*Section information type with real values*)
		Value : ARRAY[0..15]OF REAL; (*Value of the sensor*)
		Warning : ARRAY[0..15]OF BOOL; (*Temperature warning*)
		Error : ARRAY[0..15]OF BOOL; (*Temperature error*)
	END_STRUCT;
	SectionType : 	STRUCT  (*Section information type with uint values*)
		Value : ARRAY[0..15]OF UINT; (*Value of the sensor*)
		Warning : ARRAY[0..15]OF BOOL; (*Temperature warning*)
		Error : ARRAY[0..15]OF BOOL; (*Temperature error*)
		UserDisableMask : UINT; (*UserDisable mask for temperature sensors*)
		UserEnableMask : UINT; (*UserEnable mask for temperature sensors*)
		DefaultMask : UINT; (*Default mask for temperature sensors*)
		EffectiveMask : UINT; (*Effective mask for temperature sensors*)
		SensorActivated : ARRAY[0..15]OF BOOL; (*Indicates which sensors are active*)
	END_STRUCT;
END_TYPE

(*Shuttle position*)

TYPE
	ShuttlePosition : 	STRUCT  (*Actual position of the shuttle on the SuperTrak*)
		Position : DINT; (*Actual position*)
		Section : USINT; (*Actual section*)
		PositionOld : DINT; (*Position one cycle ago*)
	END_STRUCT;
	ErrorBitSectionType : 	STRUCT  (*Check if the error has been already read*)
		ErrorBitSet : ARRAY[0..31]OF BOOL; (*Check if the error has been already read*)
	END_STRUCT;
END_TYPE
```

#### Variables.var - Local variables
```iecst
(************************************************************************************************************************************)
(************************************************************************************************************************************)
(*Configuration*)
VAR CONSTANT
	CONFIG_ST_MAX_COMMANDS : USINT := 48; (*Maximum number of commands*)
	CONFIG_ST_MAX_PALLETS : USINT := 24; (*Maximum number of shuttles*)
	CONFIG_ST_MAX_SECTIONS : USINT := 4; (*Maximum number of sections*)
	CONFIG_ST_MAX_SECTIONS_MINUS_ONE : USINT := CONFIG_ST_MAX_SECTIONS-1; (*Maximum number of sections minus one*)
	CONFIG_ST_MAX_TARGETS : USINT := 48; (*Maximum number of targets*)
	CONFIG_USED_TARGETS : USINT := 6; (*Used targets on the system*)
	CONFIG_USED_TARGETS_MINUS_ONE : USINT := CONFIG_USED_TARGETS-1; (*Used targets on the system minus one*)
	CONFIG_USED_SHUTTLES : USINT := 4; (*Used shuttles on the system*)
	CONFIG_USED_SHUTTLES_MINUS_ONE : USINT := CONFIG_USED_SHUTTLES-1; (*Used shuttles on the system minus one*)
END_VAR
(************************************************************************************************************************************)
(************************************************************************************************************************************)
(*Command variable*)
VAR
	SuperTrakControl : {REDUND_UNREPLICABLE} SuperTrakCtrlType := (0); (*Variable to control the SuperTrak system*)
END_VAR
(************************************************************************************************************************************)
(************************************************************************************************************************************)
(*Function blocks*)
VAR
	StControl_0 : {REDUND_UNREPLICABLE} StControl; (*Function block to communicate to SuperTrak*)
	StSection_ : {REDUND_UNREPLICABLE} ARRAY[0..CONFIG_ST_MAX_SECTIONS_MINUS_ONE] OF StSection; (*Function blocks to control SuperTrak sections*)
	StPallet_ : {REDUND_UNREPLICABLE} ARRAY[0..CONFIG_USED_SHUTTLES_MINUS_ONE] OF StPallet; (*Function block to control shuttles*)
	StTargetExt_ : {REDUND_UNREPLICABLE} ARRAY[0..CONFIG_USED_TARGETS_MINUS_ONE] OF StTargetExt; (*Function blocks to control SuperTrak targets*)
	StAdvCmd_0 : {REDUND_UNREPLICABLE} StAdvCmd; (*Function block for AntiSloshing implementation*)
	Target_TON : {REDUND_UNREPLICABLE} ARRAY[0..CONFIG_USED_TARGETS] OF TON; (*Timer for shuttle control*)
END_VAR
(************************************************************************************************************************************)
(************************************************************************************************************************************)
(*Function block parameters*)
VAR
	SuperTrakControlParameters : {REDUND_UNREPLICABLE} StControlParType; (*Parameters for StControl*)
	SuperTrakSectionParameters : {REDUND_UNREPLICABLE} StSectionParType; (*Parameters for StSection*)
	PalletControlParameters : {REDUND_UNREPLICABLE} ARRAY[0..CONFIG_USED_SHUTTLES_MINUS_ONE] OF StPalletParType; (*Parameters for StPallet*)
	StAdvCmdParameters : {REDUND_UNREPLICABLE} StAdvCmdParType; (*Parameters for AdvancedCommand Function Block*)
	TargetControlParameters : {REDUND_UNREPLICABLE} ARRAY[0..CONFIG_USED_TARGETS_MINUS_ONE] OF StTargetExtParType; (*Parameters for each StTargetExt*)
END_VAR
(************************************************************************************************************************************)
(************************************************************************************************************************************)
(*Anti-Sloshing*)
VAR
	cmd_StartAntiSloshing : BOOL; (*Execute the Anti-Sloshing Sequence*)
	cmd_StopAntiSloshing : BOOL; (*Stop the Anti-Sloshing Sequence*)
	StopTime : TIME := T#1s; (*Time for Anti-Sloshing stillstand on target*)
	ContainerShape : USINT; (*Container shape*)
	ContainerLength : UINT; (*Lenght of the Anti-Sloshing container in mm*)
	ContainerHeight : UINT; (*Fill height of the Anti-Sloshing container in mm*)
END_VAR
(************************************************************************************************************************************)
(************************************************************************************************************************************)
(*Pallet-Control*)
VAR
	cmd_StartPalletControl : BOOL; (*Execute the PalletControl*)
	cmd_StopPalletControl : BOOL; (*Stop the PalletControl*)
END_VAR
(************************************************************************************************************************************)
(************************************************************************************************************************************)
(*Tracking*)
VAR
	cmd_StartTracking : BOOL; (*Start the Tracking fuciton*)
	cmd_StopTracking : BOOL; (*Stop the Tracking fuction*)
	StateCnc : USINT; (*State of the Tracking*)
END_VAR
VAR CONSTANT
	EXPERT_MODE_START : USINT := 0; (*Start the Expert mode*)
	EXPERT_MODE_EXECUTE : USINT := 1; (*Execute the Expert mode*)
END_VAR
VAR
	SuperTrakBeginExtCtrlStatus : BOOL; (*Status for entering the expert mode*)
	Position : DINT; (*Position of the axis to calculate shuttle position*)
END_VAR
VAR CONSTANT
	SectionLength : ARRAY[1..CONFIG_ST_MAX_SECTIONS] OF DINT := [1000000,1030000,1000000,1030000]; (*Length of every section*)
END_VAR
VAR
	CncUpdatePosition : DINT; (*Position of the shuttle on the section*)
	CncUpdateSection : USINT; (*Section where the shuttle is located*)
	CncUpdateAccel : REAL; (*Acceleration of the shuttle*)
	CncUpdateVelocity : REAL; (*Velocity of the coupled axis*)
	OldVelocity : REAL; (*Velocity to calculate the acceleration*)
	SuperTrakPalletControlStatus : BOOL; (*Tracking status*)
	CncStartTarget : USINT; (*Start Target for Cnc control*)
	ControlledShuttle : USINT; (*ID of the controlled shuttle*)
	CycleTime : REAL; (*Actual cycle time to calculate the acceleration*)
	RTInfo_0 : RTInfo; (*FUB to read the actual cycle time*)
END_VAR
(************************************************************************************************************************************)
(************************************************************************************************************************************)
(*Error handling*)
VAR
	ErrorInfo : InfoType; (*Error informations*)
END_VAR
VAR CONSTANT
	ErrorTexts : ARRAY[0..31] OF STRING[80] := ['Motor supply voltage out of range','Not specified','License not present','Not specified','Excessive coil current','High temperature','Not specified','Gateway network error','Excessive coil current(I²T)','Excessive current loop error','Not specified','Coil driver(s) shut down',2('Not specified'),'Encoder calibration required','Excessive pallet following error','Unrecognized pallet(s) detected',2('Not specified'),'Two pallets in collision deadlock','Pallet lost position feedback','Encoder read error','Coil driver error','Conflicting pallets detected','PLC Interface Heartbeat Timeout','Encoder communication error','Disabled pallet arrived','Abnormal condition detected','Section disabled through configuration software','Too many pallets','Hardware initialization error','Fatal abnormal condition detected']; (*Error texts used in TrackMaster*)
	WarningTexts : ARRAY[0..31] OF STRING[80] := [2('Application warning'),'License not present','Not specified','Thermal sensor malfunction','High temperature','Pallet position is uncertain at destination','Gateway network warning','Excessive coil current (I²T)','Coil(s) unresponsive; check connections','Not specified','Pallet position correction was required','Pallet ID tag warning','Duplicate Pallet ID detected','Two pallets in collision deadlock','Counts out of range during encoder handoff','Consecutive encoder readings out of range','Invalid region configuration','Invalid parameter configuration','Command failed','Invalid sync zone configuration','Encoder read warning','Coil driver warning','Parameter save required','Pallet destination updated','Encoder communication warning','Disabled pallet arrived','Too many pallets','Reset required to activate configuration changes','Excessive Pallet Settling Time','Controller health warning','Abnormal condition detected']; (*Warning texts used in TrackMaster*)
END_VAR
VAR
	Counter : {REDUND_UNREPLICABLE} USINT; (*Counts the errors andn warnings*)
	FaultBitCounter : USINT; (*Counts the error bit*)
	FaultBit : USINT; (*Bit that is set to get the right information*)
	WarningBit : USINT; (*Bit that is set to get the right information*)
	VisuAlarmSection : USINT; (*Actual selected section on visu*)
	VisuAlarmSectionText : ARRAY[0..23] OF STRING[80]; (*Alarm text that should be displayed in the table*)
	VisuWarningSectionText : ARRAY[0..23] OF STRING[80]; (*Warning text that should be displayed in the table*)
	AcknowledgeSelectedSection : BOOL; (*Acknowledge the selected section*)
	AcknowledgeAll : BOOL; (*Acknowledge all error*)
	CountDownAlarm : BOOL; (*Count down one section*)
	CountUpAlarm : BOOL; (*Count up one section*)
	AcknowledgeSelectedTarget : BOOL; (*Acknowledge the selected target*)
	SelectedTarget : USINT; (*Selected target on the alarm page*)
	AcknowledgeSelectedShuttle : BOOL; (*Acknowledge the selected shuttle*)
	SelectedShuttle : USINT; (*Selected shuttle on the alarm page*)
END_VAR
VAR CONSTANT
	HmiErrorTexts : ARRAY[0..15] OF STRING[80] := ['Not specified','An invalid section number was specified.','The specified parameter number was not recognized.','The specified task code was not recognized.','The requested operation is currently unavailable.','Not specified','The specified starting index is invalid.','The value to be written was outside of the valid range.','The requested number of elements is invalid.','Not specified','The command did not complete in a timely manner.','The request was denied due to a lack of permissions.',2('Not specified'),'The packet is malformed, or its length is incorrect.','An internal error occurred while processing the request.']; (*Error texts used in StHmi*)
END_VAR
VAR
	ErrorCode : UINT; (*Error code from the StHmiReadParID or StHmiWriteParID FUB*)
END_VAR
(************************************************************************************************************************************)
(************************************************************************************************************************************)
(*Read temperatures*)
VAR
	Temperatures : TemperaturesType; (*Temperatures of the SuperTrak*)
	StartIndex : USINT; (*Counter variable*)
	SectionID : USINT; (*Counter variable for the section*)
END_VAR
VAR CONSTANT
	TemperatureID : UINT := 1570; (*ID for reading temperatures*)
	WarningTemperature : REAL := 60; (*Max. temperature before warning*)
	ErrorTemperature : REAL := 80; (*Max. temperature before error*)
END_VAR
VAR
	CountDown : BOOL; (*Go to previous section*)
	CountUp : BOOL; (*Go to next section*)
	VisuSection : USINT; (*Section shown on Visu*)
	VisuTemp : RealSectionType; (*Temperatures shown on Visu*)
END_VAR
VAR CONSTANT
	MAX_SECTIONS : USINT := CONFIG_ST_MAX_SECTIONS; (*Number of sections*)
END_VAR
VAR
	i : USINT; (*Counter variable*)
END_VAR
(************************************************************************************************************************************)
(************************************************************************************************************************************)
(*Set Shuttle IDs*)
VAR
	StartTarget : USINT; (*Target where shuttles get IDs*)
	IndexSetIDs : USINT; (*Counter*)
	NumberOfShuttles : USINT; (*Number of shuttles on the SuperTrak*)
	IDSet : BOOL; (*Flag if shuttles have IDs*)
	ReleasedShuttles : USINT; (*Number of shuttles released from Wait target*)
	WaitTarget : USINT; (*Stop before shuttles go back to start position*)
END_VAR
(************************************************************************************************************************************)
(************************************************************************************************************************************)
(*Enable/Disable Region*)
VAR
	StWritePnu_Region : StWritePnu; (*Write the command to control the region*)
	StWritePnuPar_Region : StWritePnuParType; (*Parameter for StWritePnu FUB to control the region*)
	StReadPnu_Region : StReadPnu; (*Read the status of the region*)
	StReadPnuPar_Region : StReadPnuParType; (*Parameter for StReadPnu FUB to read the status of the region*)
END_VAR
VAR CONSTANT
	Region : UINT := 0; (*Command to disable the region*)
END_VAR
VAR
	RegionStatus : UINT; (*Status of the region*)
END_VAR
VAR CONSTANT
	RegionEnable : UINT := 7; (*Set the command to enable the region*)
END_VAR
VAR
	RegionEnabled : BOOL; (*The region is enabled*)
	RegionDisabled : BOOL; (*The region is disabled*)
	TimerRegionEnable : TON; (*Time before resetting the write command to enable the section*)
END_VAR
VAR CONSTANT
	Save_Parameter : UINT := 971; (*ParID to save commands*)
	SaveValue : UDINT := 8; (*Value for saving region configuration*)
END_VAR
(************************************************************************************************************************************)
(************************************************************************************************************************************)
(*Standstill check*)
VAR
	ShuttleInfo : ARRAY[0..127] OF SuperTrakPalletInfo_t; (*Actual shuttle information*)
	PositionDelta : ARRAY[0..127] OF ShuttlePosition; (*Actual, previous position and actual section*)
END_VAR
VAR CONSTANT
	PositionOffset : USINT := 100; (*Range where shuttle can be to be in standstill*)
END_VAR
VAR
	ShuttlesStandstill : BOOL; (*All shuttles are not moving*)
END_VAR
(************************************************************************************************************************************)
(************************************************************************************************************************************)
(*mappAlarmX*)
(* Function and Functionblocks *)
VAR
	MpAlarmXCore_0 : MpAlarmXCore;
	MpAlarmXHistory_0 : MpAlarmXHistory;
END_VAR
(* Structures used for HMI connection *)
VAR
	WarningStrings1 : ARRAY[0..31] OF STRING[255] := ['stw0','stw1','stw2','stw3','stw4',2('stw5'),'stw7','stw8','stw9','stw10','stw11','stw12','stw13','stw14','stw15','stw16','stw17','stw18','stw19','stw20','stw21','stw22','stw23','stw24','stw25','stw26','stw27','stw28','stw29','stw30','stw31']; (*Array that contains the error names*)
	ErrorStrings1 : ARRAY[0..31] OF STRING[255] := ['st0','st1','st2','st3','sz4','st5','st6','st7','st8','st9','st10','st11','st12','st13','st14','st15','st16','st17','st18','st19','st20','st21','st22','st23','st24','st25','st26','st27','st28','st29','st30','st31']; (*Array contains the warning names*)
	WarningStrings : ARRAY[0..31] OF STRING[255] := ['w0','w1','w2','w3','w4','w5','w6','w7','w8','w9','w10','w11','w12','w13','w14','w15','w16','w17','w18','w19','w20','w21','w22','w23','w24','w25','w26','w27','w28','w29','w30','w31']; (*Array that contains the error names*)
	ErrorStrings : ARRAY[0..31] OF STRING[255] := ['0','1','2','3','4','5','6','7','8','9','10','11','12','13','14','15','16','17','18','19','20','21','22','23','24','25','26','27','28','29','30','31']; (*Array contains the warning names*)
	counter : INT;
	Index : {REDUND_UNREPLICABLE} USINT := 0; (*Index variable used in for loops*)
	ErrorBitOnSection : ARRAY[0..CONFIG_ST_MAX_SECTIONS_MINUS_ONE] OF ErrorBitSectionType;
	WarningBitSection : ARRAY[0..CONFIG_ST_MAX_SECTIONS_MINUS_ONE] OF ErrorBitSectionType;
	SaveHistory : BOOL;
END_VAR
(************************************************************************************************************************************)
(************************************************************************************************************************************)
(*Hmi interface for read / write ParIDs*)
VAR
	HmiLink : HMILinkType; (*Link between the Hmi FUBs*)
	HmiControl_0 : HMIControl; (*HmiControl FUB to control all FUBs*)
	HmiWriteParID_0 : HMIWriteParID; (*HmiWriteParID to write ParIDs from HMI*)
	HmiReadParID_0 : HMIReadParID; (*HmiReadParID to read ParIDs from HMI*)
	HmiWritePar : HMIWriteParType; (*Parameter structure for HmiWriteParID*)
	HmiReadPar : HMIReadParType; (*Parameter structure for HmiReadParID*)
	SaveSuccessful : BOOL; (*Parameter save successful*)
	SaveFailed : BOOL; (*Parameter save failed*)
END_VAR
(************************************************************************************************************************************)
(************************************************************************************************************************************)
(*Shuttle config*)
VAR
	CountUpShuttle : BOOL; (*Count up one shuttle*)
	CountDownShuttle : BOOL; (*Count down one shuttle*)
	VisuShuttle : UINT; (*Actual shuttle*)
	Config_ShelfWidth : REAL; (*Shelf width of the shuttle*)
	Config_OffsetFromCenter : REAL; (*Offset from center from the shuttle*)
	Config_ControlGainSetIndex : USINT; (*Control gain of the shuttle*)
	Config_FilterWeightMoving : REAL; (*Filter weight moving of the shuttle*)
	Config_FilterWeightStationary : REAL; (*Filter weight stationary of the shuttle*)
	Config_SetPalletShelf : BOOL; (*Set the shuttle shelf parameters*)
	Config_SetGain : BOOL; (*Set the control gain settings*)
END_VAR
(************************************************************************************************************************************)
(************************************************************************************************************************************)
(*Other variables*)
VAR
	ReadyToReset : BOOL;
	Index2 : USINT;
END_VAR
```

#### AntiSloshing.st - Anti-Sloshing task
```iecst
(*********************************************************************************
 * Copyright: COPYRIGHT (C) BERNECKER + RAINER, AUSTRIA
 *********************************************************************************
 * Author:  B+R  Created:  November 23, 2017/08:15 PM
 *********************************************************************************
 * Description: Implementation of the AntiSloshing functionality for every shuttle
 *********************************************************************************)
ACTION AntiSloshing:
	// Execute AntiSloshing
	IF cmd_StartAntiSloshing THEN
		// Wait for shuttle
		StAdvCmdParameters.Context 				:= StTargetExt_[0].PalletID;
		StAdvCmdParameters.Parameters[0] 		:= ContainerShape;
		brsmemcpy(ADR(StAdvCmdParameters.Parameters[2]),ADR(ContainerLength),SIZEOF(ContainerLength));
		brsmemcpy(ADR(StAdvCmdParameters.Parameters[4]),ADR(ContainerHeight),SIZEOF(ContainerHeight));

		// Set proper Motion-Parameters for used container
		TargetControlParameters[0].PalletConfig.Motion.Velocity 	:= 2000;	//  [mm/s]
		TargetControlParameters[0].PalletConfig.Motion.Acceleration := 3500;	//	[mm/s²]
		//
		StTargetExt_[0].SetPalletMotionPar 		:= TRUE;
		IF	StTargetExt_[0].CommandDone THEN
			StTargetExt_[0].SetPalletMotionPar 	:= FALSE;
			// Execute the AntiSloshing
			StAdvCmd_0.SendCommand 				:= TRUE;
			cmd_StartAntiSloshing 				:= FALSE;
		END_IF;
	END_IF
	// Reset the Input of the Antisloshing function block
	IF ((EDGEPOS(StAdvCmd_0.CommandDone) AND StAdvCmd_0.SendCommand) OR StTargetExt_[0].Update OR StTargetExt_[4].Update OR StTargetExt_[5].Update) AND NOT(cmd_StopAntiSloshing)THEN
		StAdvCmd_0.SendCommand 						:= FALSE;

		// Set the Destination-Targets for each Target
		TargetControlParameters[0].AdvancedReleaseConfig.DestinationTarget := 5;
		TargetControlParameters[0].AdvancedReleaseConfig.Direction := stCOM_DIR_RIGHT;
		TargetControlParameters[4].AdvancedReleaseConfig.DestinationTarget := 6;
		TargetControlParameters[4].AdvancedReleaseConfig.Direction := stCOM_DIR_RIGHT;
		TargetControlParameters[5].AdvancedReleaseConfig.DestinationTarget := 5;
		TargetControlParameters[5].AdvancedReleaseConfig.Direction := stCOM_DIR_LEFT;

		// Update the targets
		StTargetExt_[0].Update						:= TRUE;
		StTargetExt_[4].Update						:= TRUE;
		StTargetExt_[5].Update						:= TRUE;
		IF StTargetExt_[0].UpdateDone AND StTargetExt_[4].UpdateDone AND StTargetExt_[5].UpdateDone THEN
			StTargetExt_[0].Update					:= FALSE;
			StTargetExt_[4].Update					:= FALSE;
			StTargetExt_[5].Update					:= FALSE;
			SuperTrakControl.Status.AntiSloshingEnabled := TRUE;
			StTargetExt_[0].ReleaseToTarget				:= TRUE;
		END_IF;
	END_IF
	IF StTargetExt_[0].PalletPresent = FALSE THEN
		StTargetExt_[0].ReleaseToTarget				:= FALSE;
	END_IF;
	// Timer for Stopping on the Target
	Target_TON[0].PT := StopTime;
	Target_TON[0].IN := StTargetExt_[4].PalletPresent OR StTargetExt_[5].PalletPresent;
	Target_TON[0]();

	// Sending the Pallet constantly from Target 2 to Target 3 and back
	IF SuperTrakControl.Status.AntiSloshingEnabled THEN
		StTargetExt_[4].ReleaseToTarget := StTargetExt_[4].PalletPresent AND Target_TON[0].Q;
		StTargetExt_[5].ReleaseToTarget := StTargetExt_[5].PalletPresent AND Target_TON[0].Q AND NOT(cmd_StopAntiSloshing);
	END_IF
	// Stop Executing AntiSloshing
	IF cmd_StopAntiSloshing AND (StTargetExt_[4].PalletPresent OR StTargetExt_[5].PalletPresent OR SuperTrakControl.Status.AntiSloshingEnabled = FALSE) THEN
		cmd_StartAntiSloshing 	:= FALSE;
		StAdvCmdParameters.Parameters[0] := 0;
		StAdvCmd_0.SendCommand 	:= TRUE;
		IF EDGEPOS(StAdvCmd_0.CommandDone) AND StAdvCmd_0.SendCommand THEN
			SuperTrakControl.Status.AntiSloshingEnabled := FALSE;
		END_IF
		IF SuperTrakControl.Status.AntiSloshingEnabled = FALSE THEN
			// Send back to Init Position (Target 1)
			PalletControlParameters[StAdvCmdParameters.Context-1].AdvancedReleaseConfig.DestinationTarget 	:= 1;
			PalletControlParameters[StAdvCmdParameters.Context-1].AdvancedReleaseConfig.Direction 			:= stCOM_DIR_RIGHT;
			StPallet_[StAdvCmdParameters.Context-1].ReleaseToTarget := TRUE;
			// Reset Inputs after the Pallet is in Position
			IF StPallet_[StAdvCmdParameters.Context-1].CommandDone THEN
				StPallet_[StAdvCmdParameters.Context-1].ReleaseToTarget 	:= FALSE;
				cmd_StopAntiSloshing			:= FALSE;
				StAdvCmd_0.SendCommand 			:= FALSE;
			END_IF
		END_IF
	END_IF

END_ACTION
```

#### PalletControl.st - Pallet control task
```iecst
(*****************************************************************************
 * Copyright: COPYRIGHT (C) BERNECKER + RAINER, AUSTRIA
 *****************************************************************************
 * Author:  B+R  Created:  June 21, 2017/10:34 AM
 *****************************************************************************
 * Description: Implementation of a Pallet-Control
 ******************************************************************************)
ACTION PalletControl:

	IF cmd_StartPalletControl THEN
		// Definition of the Destination-Target and the Direction of the movement
		TargetControlParameters[0].AdvancedReleaseConfig.DestinationTarget := 2;
		TargetControlParameters[0].AdvancedReleaseConfig.Direction			:= stCOM_DIR_RIGHT;
		TargetControlParameters[1].AdvancedReleaseConfig.DestinationTarget := 3;
		TargetControlParameters[1].AdvancedReleaseConfig.Direction	       := stCOM_DIR_RIGHT;
		TargetControlParameters[2].AdvancedReleaseConfig.DestinationTarget := 1;
		TargetControlParameters[2].AdvancedReleaseConfig.Direction	        := stCOM_DIR_RIGHT;

		// Change Motion-Parameters at target
		IF EDGEPOS(StTargetExt_[1].PalletPresent) THEN
			TargetControlParameters[1].PalletConfig.Motion.Acceleration := 10000;
			TargetControlParameters[1].PalletConfig.Motion.Velocity		:= 1000;
			StTargetExt_[1].SetPalletMotionPar							:= TRUE;
		END_IF
		// Reset Input after command is done
		IF EDGEPOS(StTargetExt_[1].CommandDone) AND StTargetExt_[1].SetPalletMotionPar THEN
			StTargetExt_[1].SetPalletMotionPar							:= FALSE;
		END_IF
		// Release shuttle
		IF EDGENEG(StTargetExt_[1].CommandDone) AND StTargetExt_[1].PalletPresent THEN
			StTargetExt_[1].ReleaseToTarget := TRUE;
		END_IF
		// Reset the Relase to target command
		IF NOT(StTargetExt_[1].PalletPresent) THEN
			StTargetExt_[1].ReleaseToTarget := FALSE;
		END_IF
		// Change Motion-Parameters at target
		IF EDGEPOS(StTargetExt_[2].PalletPresent) THEN
			TargetControlParameters[2].PalletConfig.Motion.Acceleration := 15000;
			TargetControlParameters[2].PalletConfig.Motion.Velocity		:= 2500;
			StTargetExt_[2].SetPalletMotionPar							:= TRUE;
		END_IF
		// Reset Input after command is done
		IF EDGEPOS(StTargetExt_[2].CommandDone) AND StTargetExt_[2].SetPalletMotionPar THEN
			StTargetExt_[2].SetPalletMotionPar							:= FALSE;
		END_IF
		IF EDGENEG(StTargetExt_[2].CommandDone) THEN
			StTargetExt_[2].ReleaseToTarget := TRUE;
		END_IF
		// Reset the Relase to target command
		IF NOT(StTargetExt_[2].PalletPresent) THEN
			StTargetExt_[2].ReleaseToTarget := FALSE;
		END_IF

		// Simple release options of the pallet for target 1
		StTargetExt_[0].ReleaseToTarget 	:= StTargetExt_[0].PalletPresent;

		// Set Status
		SuperTrakControl.Status.PalletControl	:= TRUE;
	END_IF

	// Stop pallet-control after user event
	IF cmd_StopPalletControl THEN
		cmd_StartPalletControl 	:= FALSE;
		cmd_StopPalletControl	:= FALSE;
		SuperTrakControl.Status.PalletControl	:= FALSE;
	END_IF

END_ACTION
```

#### ExpertMode.st - Expert mode task
```iecst
(*****************************************************************************
 * Copyright: COPYRIGHT (C) BERNECKER + RAINER, AUSTRIA
 *****************************************************************************
 * Author:  B+R  Created:  November 23, 2017/09:45 AM
 *****************************************************************************
 * Description: Implementation OF the Tracking functionality
 ****************************************************************************)

(*****************************************************************************)
(*****************************************************************************)
(*************************NO COLLISION AVOIDANCE******************************)
(*****************************************************************************)
(*****************************************************************************)

ACTION ExpertMode:
	(* IF all Sections are enabled the program can be executed *)
	IF SuperTrakControl.Status.AllSectionsEnabled THEN
		(* State of the Tracking *)
		CASE StateCnc OF
			(* Enter the expert mode when axis is on position = 0 to start the tracking *)
			(* The used shuttle should be on Section=1 Position=0 to start the tracking, otherwise jumps can happen *)
			(* Section=1 Position=0 --> Axis.Position = 0 *)
			EXPERT_MODE_START:
				IF gMpAxisBasic_0.Position = 0 THEN
					(* Axis ready *)
					gMpAxisBasic_0.MoveAbsolute		:= FALSE;
					gMpAxisBasic_0.Update			:= FALSE;
					(* Move all shuttles until shuttle 1 is on target 1 *)
					IF cmd_StartTracking AND StTargetExt_[CncStartTarget-1].PalletPresent THEN
						(* Enter the expert mode *)
						ControlledShuttle			:= StTargetExt_[CncStartTarget-1].PalletID;
						SuperTrakBeginExtCtrlStatus	:= SuperTrakBeginExternalControl(ControlledShuttle);
						IF SuperTrakBeginExtCtrlStatus THEN
							StateCnc				:= EXPERT_MODE_EXECUTE;
							SuperTrakControl.Status.TrackingEnabled	:= TRUE;
						END_IF
					END_IF;
					(* Move the axis to 0 *)
				ELSIF gMpAxisBasic_0.Position <> 0 THEN
					gMpAxisBasicParam.Position		:= 0;
					gMpAxisBasic_0.Update			:= TRUE;
					IF gMpAxisBasic_0.UpdateDone THEN
						gMpAxisBasic_0.MoveAbsolute	:= TRUE;
					END_IF;
				END_IF

			(* Tracking of the shuttle *)
			EXPERT_MODE_EXECUTE:
				(* Get the actual position of the axis *)
				Position							:= LREAL_TO_DINT(gMpAxisBasic_0.Position*1000);
				(* Calculate the section and position where the shutlle should be located *)
				FOR Index:=1 TO CONFIG_ST_MAX_SECTIONS DO
					IF Position - SectionLength[Index] < 0 THEN
						CncUpdateSection			:= Index;
						CncUpdatePosition			:= Position;
						EXIT;
					ELSE
						Position					:= Position - SectionLength[Index];
					END_IF
				END_FOR

				(* Calculate velocity and acceleration of the axis *)
				(* Velocity = mm/s and cycle time = ms *)
				(* mm/s / ms =  m/s²*)
				CncUpdateAccel						:= (gMpAxisBasic_0.Velocity-OldVelocity)/CycleTime;	//0.8 --> cycle time
				CncUpdateVelocity					:= REAL_TO_INT(gMpAxisBasic_0.Velocity);
				OldVelocity							:= gMpAxisBasic_0.Velocity;

				(* Call the Tracking function *)
				IF NOT(cmd_StopTracking) THEN
					SuperTrakPalletControlStatus	:= SuperTrakPalletControl(ControlledShuttle,CncUpdateSection,CncUpdatePosition,REAL_TO_INT(CncUpdateVelocity),CncUpdateAccel);
				END_IF;

				(* To exit this mode the StPallet FUB must be used to send the shuttle to a target *)
				(* After exit the expert mode, the SuperTrakBeginExternalControl must be called again *)
				IF cmd_StopTracking THEN
					(* Set parameters for controlled shuttle *)
					IF PalletControlParameters[ControlledShuttle-1].AdvancedReleaseConfig.DestinationTarget <> CncStartTarget OR PalletControlParameters[ControlledShuttle-1].AdvancedReleaseConfig.Direction <> stCOM_DIR_RIGHT THEN
						PalletControlParameters[ControlledShuttle-1].AdvancedReleaseConfig.DestinationTarget	:= CncStartTarget;
						PalletControlParameters[ControlledShuttle-1].AdvancedReleaseConfig.Direction			:= stCOM_DIR_RIGHT;
						PalletControlParameters[ControlledShuttle-1].PalletConfig.Motion.Acceleration 			:= 20000;
						PalletControlParameters[ControlledShuttle-1].PalletConfig.Motion.Velocity 				:= 2000;
						StPallet_[ControlledShuttle-1].Update			:= TRUE;
					ELSE
						StPallet_[ControlledShuttle-1].ReleaseToTarget	:= TRUE;
					END_IF;
					(* Release the shuttle *)
					IF StPallet_[ControlledShuttle-1].UpdateDone THEN
						StPallet_[ControlledShuttle-1].ReleaseToTarget	:= TRUE;
						StPallet_[ControlledShuttle-1].Update			:= FALSE;
					END_IF;
					(* Reset the parameter *)
					IF StPallet_[ControlledShuttle-1].CommandDone AND StPallet_[ControlledShuttle-1].ReleaseToTarget THEN
						StPallet_[ControlledShuttle-1].ReleaseToTarget	:= FALSE;
						StateCnc					:= EXPERT_MODE_START;
						cmd_StartTracking			:= FALSE;
						cmd_StopTracking			:= FALSE;
						gMpAxisBasic_0.MoveAbsolute	:= FALSE;
						gMpAxisBasic_0.MoveAdditive	:= FALSE;
						gMpAxisBasic_0.MoveVelocity	:= FALSE;
						gMpAxisBasic_0.JogNegative	:= FALSE;
						gMpAxisBasic_0.JogPositive	:= FALSE;
						SuperTrakControl.Status.TrackingEnabled			:= FALSE;
					END_IF;
				END_IF;

		END_CASE
	END_IF
END_ACTION
```
